PROGRAM P_Observer_Pattern
VAR
	eventPublisher					: FB_Publisher;
	eventSubscriber1				: FB_EventSubscriber1;	
	eventSubscriber2				: FB_EventSubscriber2;	
END_VAR

eventPublisher();
eventSubscriber1(eventPublisher:=eventPublisher);
eventSubscriber2(eventPublisher:=eventPublisher);

END_PROGRAM

(* stored: Version 1.1.0.1, ProductVersion 3.1.4024.11
   POU P_Observer_Pattern: Id {5faa3a49-42e7-4978-b72e-a8bc09894fca}, SpecialFunc None *)
